FUNCTION_BLOCK _SINT_TestSuite EXTENDS TcUnit.FB_TestSuite
VAR
END_VAR

TestAddress();
TestClearReference();
TestClone();
TestIecTypeReturnsExpected();
TestMakeReferenceToFollowsReference();
TestMakeReferenceToUpdatesReference();
TestSize();
TestValueReturnsExpectedAfterInit();
TestValueReturnsExpectedAfterChange();
TestSerializeTypeWith();
TestSerializeWith();
TestTryDeserializeFrom();
TestTryMakeReferenceToFollowsReference();
TestTryMakeReferenceToUpdatesReference();

METHOD PUBLIC TestAddress
VAR
    _type : _SINT(0);
    notExpected : PVOID := 0;
    actual : PVOID;
END_VAR
TEST('TestAddress');

actual := _type.Address;

AssertFalse(
    Condition := (notExpected = actual),
    Message := 'Type did not return a valid address.'
);

TEST_FINISHED();
END_METHOD

METHOD PUBLIC TestClearReference
VAR
    _type : _SINT(0);
	target : SINT := 0;
    expected : SINT := 0;
    actual : SINT;
END_VAR
TEST('TestClearReference');

_type.MakeReferenceTo(target);
_type.ClearReference();
target := 123;

actual := _type.Value;

AssertEquals(
    Expected := expected,
    Actual := actual,
    Message := 'Value did not follow target change'
);

TEST_FINISHED();
END_METHOD

METHOD PUBLIC TestClone
VAR
    _type : _SINT(123);
	clone : I_Datatype;
	isValidClone : BOOL;
	compareResult : DINT;
END_VAR
TEST('TestClone');

clone := _type.Clone();

isValidClone := clone <> 0;

IF isValidClone THEN
	compareResult := memcmp(_type.Address, clone.Address, clone.Size);
END_IF

AssertTrue(
	Condition := isValidClone,
	Message := 'Clone did not produce a clone'
);

AssertEquals_DINT(
	Expected := 0,
    Actual := compareResult,
    Message := 'Clone did not return a valid clone.'
);

clone.Dispose();

TEST_FINISHED();
END_METHOD

METHOD PUBLIC TestIecTypeReturnsExpected
VAR
    _type : _SINT(0);
    expected : STRING := 'SINT';
    actual : STRING;
END_VAR
TEST('TestIecTypeReturnsExpected');

actual := _type.IecType;

AssertEquals_STRING(
    Expected := expected,
    Actual := actual,
    Message := 'Type did not return correct iec type.'
);

TEST_FINISHED();
END_METHOD

METHOD PUBLIC TestMakeReferenceToFollowsReference
VAR
    _type : _SINT(0);
	target : SINT := 0;
    expected : SINT := 123;
    actual : SINT;
END_VAR
TEST('TestMakeReferenceToFollowsReference');

_type.MakeReferenceTo(target);
target := 123;

actual := _type.Value;

AssertEquals(
    Expected := expected,
    Actual := actual,
    Message := 'Value did not follow target change'
);

TEST_FINISHED();
END_METHOD

METHOD PUBLIC TestMakeReferenceToUpdatesReference
VAR
    _type : _SINT(0);
	target : SINT := 0;
    expected : SINT := 123;
    actual : SINT;
END_VAR
TEST('TestMakeReferenceToUpdatesReference');

_type.MakeReferenceTo(target);
_type.Value := 123;

actual := target;

AssertEquals(
    Expected := expected,
    Actual := actual,
    Message := 'Value did not update target'
);

TEST_FINISHED();
END_METHOD

METHOD PUBLIC TestSerializeTypeWith
VAR
    _type : _SINT(0);
    serializer : JsonSerializer;
    expected : STRING := '{"type":"SINT"}';
    actual : STRING(500);
END_VAR
TEST('TestSerializeTypeWith');

serializer.Reset();
_type.SerializeTypeWith(serializer);
serializer.TryGetSerializedData(ADR(actual), SIZEOF(actual));

AssertEquals_STRING(
    Expected := expected,
    Actual := actual,
    Message := 'Serialization of type did not return correct string.'
);

TEST_FINISHED();
END_METHOD

METHOD PUBLIC TestSerializeWith
VAR
    _type : _SINT(123);
    serializer : JsonSerializer;
    expected : STRING := '123';
    actual : STRING(500);
END_VAR
TEST('TestSerializeWith');

serializer.Reset();
_type.SerializeWith(serializer);
serializer.TryGetSerializedData(ADR(actual), SIZEOF(actual));

AssertEquals_STRING(
    Expected := expected,
    Actual := actual,
    Message := 'Serialization of type data did not return correct string.'
);

TEST_FINISHED();
END_METHOD

METHOD PUBLIC TestSize
VAR
    _type : _SINT(0);
    expected : UDINT := SIZEOF(SINT);
    actual : UDINT;
END_VAR
TEST('TestSize');

actual := _type.Size;

AssertEquals_UDINT(
    Expected := Expected,
    Actual := actual,
    Message := 'Type did not return the correct size.'
);

TEST_FINISHED();
END_METHOD

METHOD PUBLIC TestTryDeserializeFrom
VAR
    deserializer : JsonDeserializer;
    feedback : DeserializerFeedback;
    json : STRING := '123';
    _type : _SINT(0);
    expected : SINT := 123;
    actual : SINT;
 END_VAR
TEST('TestTryDeserializeFrom');

deserializer.Reset();
deserializer.TryLoad(json);
_type.TryDeserializeFrom(Deserializer, Feedback);

actual := _type.Value;

AssertEquals(
    Expected := expected,
    Actual := actual,
    Message := 'Type did not deserialize correctly.'
);

TEST_FINISHED();
END_METHOD

METHOD PUBLIC TestTryMakeReferenceToFollowsReference
VAR
    _type : _SINT(0);
	target : _SINT(0);
    expected : SINT := 123;
    actual : SINT;
END_VAR
TEST('TestTryMakeReferenceToFollowsReference');

_type.TryMakeReferenceTo(target);
target.Value := 123;

actual := _type.Value;

AssertEquals(
    Expected := expected,
    Actual := actual,
    Message := 'Value did not follow target change'
);

TEST_FINISHED();
END_METHOD

METHOD PUBLIC TestTryMakeReferenceToUpdatesReference
VAR
    _type : _SINT(0);
	target : _SINT(0);
    expected : SINT := 123;
    actual : SINT;
END_VAR
TEST('TestTryMakeReferenceToUpdatesReference');

_type.TryMakeReferenceTo(target);
_type.Value := 123;

actual := target.Value;

AssertEquals(
    Expected := expected,
    Actual := actual,
    Message := 'Value did not update target'
);

TEST_FINISHED();
END_METHOD

METHOD PUBLIC TestValueReturnsExpectedAfterChange
VAR
    _type : _SINT(0);
    expected : SINT := 123;
    actual : SINT;
END_VAR
TEST('TestValueReturnsExpectedAfterChange');

_type.Value := 123;

actual := _type.Value;

AssertEquals(
    Expected := expected,
    Actual := actual,
    Message := 'Expected value not returned after change.'
);

TEST_FINISHED();
END_METHOD

METHOD PUBLIC TestValueReturnsExpectedAfterInit
VAR
    _type : _SINT(123);
    expected : SINT := 123;
    actual : SINT;
END_VAR
TEST('TestValueReturnsExpectedAfterInit');

actual := _type.Value;

AssertEquals(
    Expected := expected,
    Actual := actual,
    Message := 'Expected value not returned after Init.'
);

TEST_FINISHED();
END_METHOD

END_FUNCTION_BLOCK

(* stored: Version 1.1.0.1, ProductVersion 3.1.4024.12
   POU _SINT_TestSuite: Id {8253f6d9-6b74-08e1-18f9-83ade23add23}, SpecialFunc None
   Method TestAddress: Id {4afcb581-a779-008b-20ba-4a6e494e7716}
   Method TestClearReference: Id {b02dd206-0642-03d2-0945-5db0c72dc1f4}
   Method TestClone: Id {d8d9d9ea-3611-0ddf-1bae-2a2e5a6a585c}
   Method TestIecTypeReturnsExpected: Id {1d902baa-bf95-023e-0871-3befab668145}
   Method TestMakeReferenceToFollowsReference: Id {5f795c7b-5a03-0806-089d-785656fe6a8a}
   Method TestMakeReferenceToUpdatesReference: Id {c3d2938a-7e22-0f14-1d3a-c15ed8d14646}
   Method TestSerializeTypeWith: Id {d556bfa3-6e00-0886-1c90-24dc5489f380}
   Method TestSerializeWith: Id {74f12ab2-5194-02c4-3c96-303641719ee9}
   Method TestSize: Id {2bb39c24-1232-0024-139b-ed8dd946c1f2}
   Method TestTryDeserializeFrom: Id {75088590-5e60-0e69-2db0-2b319784c430}
   Method TestTryMakeReferenceToFollowsReference: Id {29820776-108e-00d3-0f7b-9a527d837896}
   Method TestTryMakeReferenceToUpdatesReference: Id {f0887213-7ddf-05c7-232a-fd51b04d78eb}
   Method TestValueReturnsExpectedAfterChange: Id {88f6dc4c-c05f-080c-19b4-5c4182b33e88}
   Method TestValueReturnsExpectedAfterInit: Id {f6808052-aca9-0ed3-0b95-93e55756ea43} *)
